// Mitsubishi GX Works2 project: GX W2 L3 Ex 1 DK C   PLC: FX3G

// global labels: Global1
VAR_GLOBAL
  iStart_PB AT X001 : BOOL;
  iStop_PB AT X002 : BOOL;
  iProx_Sensor AT X003 : BOOL;
  oConveyor AT Y000 : BOOL;
  iReset_PB AT X004 : BOOL;
  oProduct_Low AT Y001 : BOOL;
  oProduct_Full AT Y002 : BOOL;
END_VAR

// task Task_01 (event TRUE, interval 0, priority 31): POU_01

PROGRAM POU_01
VAR
  bSystem_Started : BOOL;
  CTU_1_Product_Count : CTU;
  bPause_Conveyor : BOOL;
END_VAR
(* structured ladder/FBD written out as ST: instructions are called as NAME(EN, inputs, outputs); _pN, _eN, _tN stand for wires *)
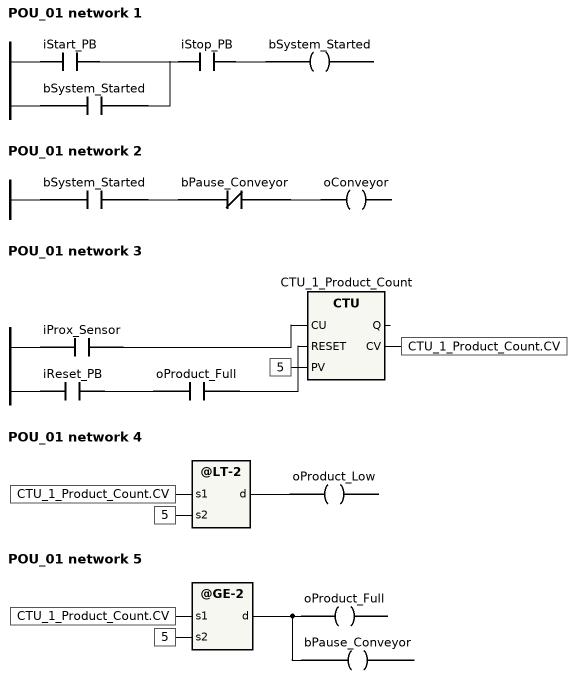
(* network 1 *)
bSystem_Started := (iStart_PB OR bSystem_Started) AND iStop_PB;
(* network 2 *)
oConveyor := bSystem_Started AND NOT bPause_Conveyor;
(* network 3 *)
CTU_1_Product_Count(CU := iProx_Sensor, RESET := iReset_PB AND oProduct_Full, PV := 5, CV => CTU_1_Product_Count.CV);
(* network 4 *)
oProduct_Low := @LT-2(CTU_1_Product_Count.CV, 5);
(* network 5 *)
_p1 := @GE-2(CTU_1_Product_Count.CV, 5);
oProduct_Full := _p1;
bPause_Conveyor := _p1;
END_PROGRAM
